// TIA Portal V16 export
// export: Created 2024-12-03T15:41:43.8995519Z, ExportSetting WithDefaults, DisplayName Totally Integrated Automation Portal, DisplayVersion V16 Update 6, DisplayName TIA Portal Version Control Interface, DisplayVersion V16 Update 2, DisplayName TIA Portal Openness, DisplayVersion V16 Update 6, DisplayName TIA Portal Teamcenter Gateway, DisplayVersion V16, DisplayName SINAMICS Startdrive Advanced, DisplayVersion V16 Update 5, DisplayName SINAMICS Startdrive G130, G150, S120, S150, SINAMICS MV, S210, DisplayVersion V16 Update 5, DisplayName SINAMICS Startdrive G110M, G120, G120C, G120D, G120P, G115D, DisplayVersion V16 Update 5, DisplayName STEP 7 Professional, DisplayVersion V16 Update 6, DisplayName STEP 7 Safety, DisplayVersion V16, DisplayName WinCC Advanced / Unified PC, DisplayVersion V16 Update 6
DATA_BLOCK "ApplicationState_DB"   // DB13
{ S7_Optimized_Access := 'FALSE' }
VERSION : 0.1
// stored: AutoNumber true, DBAccessibleFromOPCUA true, IsOnlyStoredInLoadMemory false, IsWriteProtectedInAS false
   VAR
      GlobalState : "GlobalApplicationStatus_UDT";
      Appstate { S7_SetPoint := 'True'} : Array[0..52] of "ApplicationState_UDT";
      ZoneNames { S7_SetPoint := 'True'} : Array[0..52] of "ZoneInfo";
      MasterSpeed { S7_SetPoint := 'True'} : Real;   // 50|75|100
   END_VAR
BEGIN
   GlobalState.LED.GreenLED := FALSE;
   GlobalState.LED.GreenLEDFlash := FALSE;
   GlobalState.LED.RedLED := FALSE;
   GlobalState.LED.RedLEDFlash := FALSE;
   GlobalState.LED.BlueLED := FALSE;
   GlobalState.LED.BlueLEDFlash := FALSE;
   GlobalState.States.AutoMode := FALSE;
   GlobalState.States.ManualMode := FALSE;
   GlobalState.States.EmptyMode := FALSE;
   GlobalState.States.AlarmActive := FALSE;
   GlobalState.States.EmergencyOk := FALSE;
   Appstate[0].Hmi_Buttons.reset.SignalFromHMI := FALSE;
   Appstate[0].Hmi_Buttons.reset.state.State := FALSE;
   Appstate[0].Hmi_Buttons.reset.state.LE := FALSE;
   Appstate[0].Hmi_Buttons.reset.state.FE := FALSE;
   Appstate[0].Hmi_Buttons.reset.colorNumber := 0;
   Appstate[0].Hmi_Buttons.reset.Hide := FALSE;
   Appstate[0].Hmi_Buttons.StartAutoMode.SignalFromHMI := FALSE;
   Appstate[0].Hmi_Buttons.StartAutoMode.state.State := FALSE;
   Appstate[0].Hmi_Buttons.StartAutoMode.state.LE := FALSE;
   Appstate[0].Hmi_Buttons.StartAutoMode.state.FE := FALSE;
   Appstate[0].Hmi_Buttons.StartAutoMode.colorNumber := 0;
   Appstate[0].Hmi_Buttons.StartAutoMode.Hide := FALSE;
   Appstate[0].Hmi_Buttons.ActivateManualMode.SignalFromHMI := FALSE;
   Appstate[0].Hmi_Buttons.ActivateManualMode.state.State := FALSE;
   Appstate[0].Hmi_Buttons.ActivateManualMode.state.LE := FALSE;
   Appstate[0].Hmi_Buttons.ActivateManualMode.state.FE := FALSE;
   Appstate[0].Hmi_Buttons.ActivateManualMode.colorNumber := 0;
   Appstate[0].Hmi_Buttons.ActivateManualMode.Hide := FALSE;
   Appstate[0].Hmi_Buttons.StopAutoMode.SignalFromHMI := FALSE;
   Appstate[0].Hmi_Buttons.StopAutoMode.state.State := FALSE;
   Appstate[0].Hmi_Buttons.StopAutoMode.state.LE := FALSE;
   Appstate[0].Hmi_Buttons.StopAutoMode.state.FE := FALSE;
   Appstate[0].Hmi_Buttons.StopAutoMode.colorNumber := 0;
   Appstate[0].Hmi_Buttons.StopAutoMode.Hide := FALSE;
   Appstate[0].Hmi_Buttons.DeactivateManualMode.SignalFromHMI := FALSE;
   Appstate[0].Hmi_Buttons.DeactivateManualMode.state.State := FALSE;
   Appstate[0].Hmi_Buttons.DeactivateManualMode.state.LE := FALSE;
   Appstate[0].Hmi_Buttons.DeactivateManualMode.state.FE := FALSE;
   Appstate[0].Hmi_Buttons.DeactivateManualMode.colorNumber := 0;
   Appstate[0].Hmi_Buttons.DeactivateManualMode.Hide := FALSE;
   Appstate[0].Hmi_Buttons.StartEmptyMode.SignalFromHMI := FALSE;
   Appstate[0].Hmi_Buttons.StartEmptyMode.state.State := FALSE;
   Appstate[0].Hmi_Buttons.StartEmptyMode.state.LE := FALSE;
   Appstate[0].Hmi_Buttons.StartEmptyMode.state.FE := FALSE;
   Appstate[0].Hmi_Buttons.StartEmptyMode.colorNumber := 0;
   Appstate[0].Hmi_Buttons.StartEmptyMode.Hide := FALSE;
   Appstate[0].Hmi_Buttons.StopEmptyMode.SignalFromHMI := FALSE;
   Appstate[0].Hmi_Buttons.StopEmptyMode.state.State := FALSE;
   Appstate[0].Hmi_Buttons.StopEmptyMode.state.LE := FALSE;
   Appstate[0].Hmi_Buttons.StopEmptyMode.state.FE := FALSE;
   Appstate[0].Hmi_Buttons.StopEmptyMode.colorNumber := 0;
   Appstate[0].Hmi_Buttons.StopEmptyMode.Hide := FALSE;
   Appstate[0].Hmi_Buttons.ActivateStandby.SignalFromHMI := FALSE;
   Appstate[0].Hmi_Buttons.ActivateStandby.state.State := FALSE;
   Appstate[0].Hmi_Buttons.ActivateStandby.state.LE := FALSE;
   Appstate[0].Hmi_Buttons.ActivateStandby.state.FE := FALSE;
   Appstate[0].Hmi_Buttons.ActivateStandby.colorNumber := 0;
   Appstate[0].Hmi_Buttons.ActivateStandby.Hide := FALSE;
   Appstate[0].States.ReadyForAutoMode := FALSE;
   Appstate[0].States.ReadyForStandby := FALSE;
   Appstate[0].States.RequestingAutoModeOff := FALSE;
   Appstate[2].States.ManualModeActivated.State := TRUE;
   Appstate[2].States.EmergencyOk.State := TRUE;
   Appstate[0].Alarms.AlarmActiveInternalPLC := FALSE;
   Appstate[0].Alarms.AlarmsActiveForHmi := FALSE;
   ZoneNames[0].AppStateIndex := 0;
   ZoneNames[1].AppStateIndex := 1;
   ZoneNames[2].AppStateIndex := 2;
   ZoneNames[3].AppStateIndex := 3;
   ZoneNames[4].AppStateIndex := 4;
   ZoneNames[5].AppStateIndex := 5;
   ZoneNames[6].AppStateIndex := 6;
   ZoneNames[7].AppStateIndex := 7;
   ZoneNames[8].AppStateIndex := 8;
   ZoneNames[9].AppStateIndex := 9;
   ZoneNames[10].AppStateIndex := 10;
   ZoneNames[11].AppStateIndex := 11;
   ZoneNames[12].AppStateIndex := 12;
   ZoneNames[13].AppStateIndex := 13;
   ZoneNames[14].AppStateIndex := 14;
   ZoneNames[15].AppStateIndex := 15;
   ZoneNames[16].AppStateIndex := 16;
   ZoneNames[17].AppStateIndex := 17;
   ZoneNames[18].AppStateIndex := 18;
   ZoneNames[19].AppStateIndex := 19;
   ZoneNames[20].AppStateIndex := 20;
   ZoneNames[21].AppStateIndex := 21;
   ZoneNames[22].AppStateIndex := 22;
   ZoneNames[23].AppStateIndex := 23;
   ZoneNames[24].AppStateIndex := 24;
   ZoneNames[25].AppStateIndex := 25;
   ZoneNames[26].AppStateIndex := 26;
   ZoneNames[27].AppStateIndex := 27;
   ZoneNames[28].AppStateIndex := 28;
   ZoneNames[29].AppStateIndex := 29;
   ZoneNames[30].AppStateIndex := 30;
   ZoneNames[31].AppStateIndex := 31;
   ZoneNames[32].AppStateIndex := 32;
   ZoneNames[40].AppStateIndex := 40;
   ZoneNames[41].AppStateIndex := 41;
   ZoneNames[42].AppStateIndex := 42;
   ZoneNames[43].AppStateIndex := 43;
   ZoneNames[44].AppStateIndex := 44;
   ZoneNames[45].AppStateIndex := 45;
   ZoneNames[46].AppStateIndex := 46;
   ZoneNames[47].AppStateIndex := 47;
   ZoneNames[48].AppStateIndex := 48;
   ZoneNames[49].AppStateIndex := 49;
   ZoneNames[50].AppStateIndex := 50;
   ZoneNames[51].AppStateIndex := 51;
   ZoneNames[52].AppStateIndex := 52;
   ZoneNames[0].ZoneName := 'MAIN';
   ZoneNames[10].ZoneName := 'ZONE 100 A';
   ZoneNames[11].ZoneName := 'OUTB LVL1 B';
   ZoneNames[12].ZoneName := 'OUTB LVL1 C';
   ZoneNames[13].ZoneName := 'OUTB LVL1 D';
   ZoneNames[20].ZoneName := 'ZONE 200A';
   ZoneNames[21].ZoneName := 'ZONE 200B';
   ZoneNames[22].ZoneName := 'ZONE 200C';
   ZoneNames[23].ZoneName := 'ZONE 200D';
   ZoneNames[24].ZoneName := 'ZONE 200E';
   ZoneNames[25].ZoneName := 'ZONE 200F';
   ZoneNames[26].ZoneName := 'ZONE 200G';
   ZoneNames[27].ZoneName := 'ZONE 200H';
   ZoneNames[30].ZoneName := 'ZONE 300A';
   ZoneNames[31].ZoneName := 'ZONE 300B';
   ZoneNames[32].ZoneName := 'ZONE 300C';
   ZoneNames[40].ZoneName := 'ZONE 400A';
   ZoneNames[41].ZoneName := 'INB LVL2 B';
   ZoneNames[42].ZoneName := 'INB LVL2 C';
   ZoneNames[43].ZoneName := 'INB LVL2 D';
   ZoneNames[50].ZoneName := 'ZONE_500A';
   ZoneNames[51].ZoneName := 'ZONE_500B';
   ZoneNames[52].ZoneName := 'ZONE_500C';
END_DATA_BLOCK
